// TIA Portal V16 export
// export: Created 2020-03-17T19:26:51.0293779Z, ExportSetting None, DisplayName Totally Integrated Automation Portal, DisplayVersion V16, DisplayName TIA Portal Version Control Interface, DisplayVersion V16, DisplayName TIA Portal Openness, DisplayVersion V16, DisplayName STEP 7 Professional, DisplayVersion V16, DisplayName STEP 7 Safety, DisplayVersion V16, DisplayName WinCC Advanced, DisplayVersion V16
TYPE "Step"
   STRUCT
      Next : Int;   // next step no.
      Abort : Int;   // abort step no.
      Option1 : Int;   // optional step 1
      Option2 : Int;   // optional step 2
      MonitorTime : Int;   // max. time step
      "Name" : WString[20];   // name of the step
      WaitingTime : DInt;   // wainting time
   END_STRUCT;
END_TYPE
